TYPE E_Typ_MOD :
(
	///no usage until yet
	Default := 0,
	Max_E_Typ_CYL
);
END_TYPE

(* stored: Version 1.1.0.1, ProductVersion 3.1.0.25
   DUT E_Typ_MOD: Id {9f05c469-10c2-4ea8-a9ad-a33ba5807ca8} *)
